FUNCTION_BLOCK FB_StackerLiftControl
VAR_INPUT
	FunctionData			: ST_FunctionData; 						// Function data
	ZoneData				: ST_ZoneData;
	EnableDrive				: BOOL;								//forks not moving	
	OrderPos				: E_StackerLiftPositions; 		// Order position of palletmagazine	
	LiftEncoderType			: BOOL;								// TRUE: Encoder is used for positioning, False: Inductive sensors is used
	SensorInputs			: ST_StackerLiftSensorInp;			// Lift sensor inputs
	ManualInputs			: ST_StackerLiftManualInp;			// Manual control inputs
	EncoderSettings			: ST_LSPM_LiftEncPos;			// Encoder configuration
	TimeoutValueLift		: TIME; 							// Timeout value for turning	
	
END_VAR

VAR_OUTPUT
	DriveUp					: BOOL; 							// Drive run command lift up
	DriveDown				: BOOL; 							// Drive run command lift down
	DriveCS					: BOOL; 							// Drive run command lift low speed
	EnableTransport			: BOOL;								// Enable transport
	ActualPosition			: E_StackerLiftPositions;		// The position of the lift
END_VAR

VAR_IN_OUT
	ErrorData 				: ST_ErrorDataSet; // Error data
END_VAR

VAR
	eState					: E_StackerLiftStates;
	eLastState				: E_StackerLiftStates;	
	TimerTimeoutLift		: TON;		
	TimerIdle				: TON := (PT:= T#500MS);  // delay setting EnableTransport until lift motor realy stopped
END_VAR


F_ResetError(
	Reset 	  := FALSE,
	ErrorData := ErrorData);


// Initialise variables	
DriveUp := FALSE;
DriveDown := FALSE;
EnableTransport := FALSE;	
TimerTimeoutLift.IN := FALSE;
TimerTimeoutLift.PT := TimeoutValueLift;
//ActualPosition := E_PositionsPalletMagazineForkLift.UNDEFINED;
ActualPosition 	:= _M_GetActualPosition(LiftEncoderType,SensorInputs,EncoderSettings,ErrorData);
 

CASE eState OF
	(*************************************************************************
	  Initialise
	*************************************************************************)	
	E_StackerLiftStates.INIT:
		DriveUp := FALSE;
		DriveDown := FALSE;
		DriveCS := FALSE;		
		EnableTransport := FALSE;	
	
		eLastState := eState;
		eState := E_StackerLiftStates.IDLE;
		
	(*************************************************************************
	  Error
	*************************************************************************)	
	E_StackerLiftStates.Error:

		IF NOT ManualInputs.SwitchManualAuto THEN
			eLastState := eState;
			eState := E_StackerLiftStates.MANUAL;

		// Acknowledge request error
		ELSIF ErrorData.ErrorType <> E_ErrorType.ERROR AND 
			FunctionData.ErrorData.Error.ErrorType <> E_ErrorType.ERROR AND ZoneData.ErrorData.ErrorState <> E_ErrorState.ERROR  THEN	
			eLastState := eState;
			eState := E_StackerLiftStates.Init;			
		END_IF	

	(*************************************************************************
	  Manual
	*************************************************************************)			
	E_StackerLiftStates.MANUAL:		
		IF ManualInputs.SwitchManualAuto THEN
			eLastState := eState;
			eState := E_StackerLiftStates.INIT;		
		ELSE
			_M_ManualMode(LiftEncoderType,SensorInputs,ManualInputs,EncoderSettings,ActualPosition);			
		END_IF
	(*************************************************************************
	  Idle
	*************************************************************************)		
	E_StackerLiftStates.IDLE:
		IF NOT ManualInputs.SwitchManualAuto THEN
			eLastState := eState;
			eState := E_StackerLiftStates.MANUAL;

		// If function is started and no error	
		ELSIF ((FunctionData.OperationState.eState = E_PositionState.STARTED OR FunctionData.OperationState.eState = E_PositionState.STOPPING) AND
		  	   FunctionData.ErrorData.Error.ErrorType <> E_ErrorType.ERROR AND ZoneData.ErrorData.ErrorState <> E_ErrorState.ERROR) THEN		  	
					
			DriveCS := FALSE;	
	
			IF OrderPos = E_StackerLiftPositions.DOWN THEN
				// When Lift is in position down (lowest position)
				IF ActualPosition = E_StackerLiftPositions.DOWN THEN
					EnableTransport := TimerIdle.Q;
				ELSIF(EnableDrive AND FunctionData.OperationState.eState = E_PositionState.STARTED) THEN //only start movment if group is started and not stopping
					eLastState := eState;
					eState := E_StackerLiftStates.LIFT_DOWN;
				END_IF
				
			ELSIF OrderPos = E_StackerLiftPositions.UP THEN
				// When lift is in upper position, second pallet lifted up
				IF ActualPosition = E_StackerLiftPositions.Up THEN
					EnableTransport := TimerIdle.Q;
				ELSIF(EnableDrive AND FunctionData.OperationState.eState = E_PositionState.STARTED) THEN //only start movment if group is started and not stopping
					eLastState := eState;
					eState := E_StackerLiftStates.LIFT_UP;
				END_IF
				
			ELSIF OrderPos = E_StackerLiftPositions.MIDDLE THEN
				// When lift is ordered to the middle position 
				IF ActualPosition = E_StackerLiftPositions.MIDDLE THEN
					EnableTransport := TimerIdle.Q;
				ELSIF(EnableDrive AND FunctionData.OperationState.eState = E_PositionState.STARTED) THEN //only start movment if group is started and not stopping
					IF( _M_DecideNextMovement(OrderPos,LiftEncoderType,SensorInputs,EncoderSettings) = E_StackerLiftStates.LIFT_MIDDLE_FROM_DOWN) THEN
						eLastState := eState;
						eState := E_StackerLiftStates.LIFT_MIDDLE_FROM_DOWN;
					ELSIF( _M_DecideNextMovement(OrderPos,LiftEncoderType,SensorInputs,EncoderSettings) = E_StackerLiftStates.LIFT_MIDDLE_FROM_UP) THEN
						eLastState := eState;
						eState := E_StackerLiftStates.LIFT_MIDDLE_FROM_UP;
					ELSE
						//can not decide next movment, since we dont know where we are
						F_SetError( ErrorType := E_ErrorType.ERROR, 
									ErrorParam := 'Middle position unknown.', //Can not decide next movment 
									ErrorMsg := E_ErrorConv.INCORRECT_SENSOR_SIGNAL, 
									ErrorData := ErrorData);
						
					END_IF
				END_IF			
			END_IF
		ELSE
			eLastState := eState;
			eState := E_StackerLiftStates.Error;		  
		END_IF	
	
	(*************************************************************************
	  Turn to ccw
	*************************************************************************)	
	E_StackerLiftStates.LIFT_DOWN:
		// If function is started or stopping and no error
		IF (FunctionData.OperationState.eState = E_PositionState.STARTED OR FunctionData.OperationState.eState = E_PositionState.STOPPING) AND
		  FunctionData.ErrorData.Error.ErrorType <> E_ErrorType.ERROR AND ZoneData.ErrorData.ErrorState <> E_ErrorState.ERROR THEN
			// Moving lift down until desired level is reached			
			TimerTimeoutLift.IN := TRUE;
			// If time is up
			IF TimerTimeoutLift.Q THEN
				DriveDown := FALSE;
				F_SetError(
					ErrorType := E_ErrorType.ERROR, 
					ErrorParam := 'Timeout Lifting Down', 
					ErrorMsg := E_ErrorConv.TIMEOUT_MOVEMENT, 
					ErrorData := ErrorData);
					
				eLastState := eState;
				eState := E_StackerLiftStates.Error;
			ELSIF(_M_DecideStopAndCreep(eState,LiftEncoderType,SensorInputs,EncoderSettings, ActualPosition,ErrorData,DriveCS)) THEN
				eLastState := eState;
				eState := E_StackerLiftStates.IDLE;			
			ELSIF EnableDrive THEN
				DriveDown := TRUE;
				//DriveCS := _M_DecideCreepSpeed(eState,LiftType,SensorInputs,EncoderSettings);		
			END_IF
		ELSE
			eLastState := eState;
			eState := E_StackerLiftStates.Error;			
		END_IF
		
	
	(*************************************************************************
	  Turn to cw
	*************************************************************************)		
	E_StackerLiftStates.LIFT_UP:
	
		IF (FunctionData.OperationState.eState = E_PositionState.STARTED OR FunctionData.OperationState.eState = E_PositionState.STOPPING) AND
		  FunctionData.ErrorData.Error.ErrorType <> E_ErrorType.ERROR AND ZoneData.ErrorData.ErrorState <> E_ErrorState.ERROR THEN
			// Moving lift up until desired level is reached
			TimerTimeoutLift.IN := TRUE;
				
			// If time is up
			IF TimerTimeoutLift.Q THEN
				DriveUp := FALSE;
				F_SetError(
					ErrorType := E_ErrorType.ERROR, 
					ErrorParam := 'Timeout Lifting Up', 
					ErrorMsg := E_ErrorConv.TIMEOUT_MOVEMENT, 
					ErrorData := ErrorData);
					
				eLastState := eState;
				eState := E_StackerLiftStates.Error;
			ELSIF(_M_DecideStopAndCreep(eState,LiftEncoderType,SensorInputs,EncoderSettings, ActualPosition,ErrorData,DriveCS)) THEN
				eLastState := eState;
				eState := E_StackerLiftStates.IDLE;
			ELSIF EnableDrive THEN
				DriveUp := TRUE;
				//DriveCS := _M_DecideCreepSpeed(eState,LiftType,SensorInputs,EncoderSettings);		
			END_IF		
		ELSE
			eLastState := eState;
			eState := E_StackerLiftStates.Error;			
		END_IF

	(*************************************************************************
	  Turn to middle from ccw
	*************************************************************************)
	E_StackerLiftStates.LIFT_MIDDLE_FROM_DOWN:
	
		IF (FunctionData.OperationState.eState = E_PositionState.STARTED OR FunctionData.OperationState.eState = E_PositionState.STOPPING) AND
		  FunctionData.ErrorData.Error.ErrorType <> E_ErrorType.ERROR AND ZoneData.ErrorData.ErrorState <> E_ErrorState.ERROR THEN			
			// Moving lift up to the middle poistition until desired level is reached
			TimerTimeoutLift.IN := TRUE;				
			// If time is up
			IF TimerTimeoutLift.Q THEN
				DriveUp := FALSE;
				F_SetError(
					ErrorType := E_ErrorType.ERROR, 
					ErrorParam := 'Timeout Lifting to Middle from Down', 
					ErrorMsg := E_ErrorConv.TIMEOUT_MOVEMENT, 
					ErrorData := ErrorData);
					
				eLastState := eState;
				eState := E_StackerLiftStates.Error;
			ELSIF(_M_DecideStopAndCreep(eState,LiftEncoderType,SensorInputs,EncoderSettings, ActualPosition,ErrorData,DriveCS)) THEN
				eLastState := eState;
				eState := E_StackerLiftStates.IDLE;
			ELSIF EnableDrive THEN
				DriveUp := TRUE;
				//DriveCS := _M_DecideCreepSpeed(eState,LiftType,SensorInputs,EncoderSettings);	
			END_IF

		ELSE
			eLastState := eState;
			eState := E_StackerLiftStates.Error;
		END_IF
		
	(*************************************************************************
	  Turn to middle from cw
	*************************************************************************)		
	E_StackerLiftStates.LIFT_MIDDLE_FROM_UP:
	
		IF (FunctionData.OperationState.eState = E_PositionState.STARTED OR FunctionData.OperationState.eState = E_PositionState.STOPPING) AND
		  FunctionData.ErrorData.Error.ErrorType <> E_ErrorType.ERROR AND ZoneData.ErrorData.ErrorState <> E_ErrorState.ERROR THEN			
			// Moving lift down to the middle poistition until desired level is reached
			TimerTimeoutLift.IN := TRUE;
			// If time is up
			IF TimerTimeoutLift.Q THEN
				DriveDown := FALSE;
				F_SetError(
					ErrorType := E_ErrorType.ERROR, 
					ErrorParam := 'Timeout Liftning to Middle from Up', 
					ErrorMsg := E_ErrorConv.TIMEOUT_MOVEMENT, 
					ErrorData := ErrorData);
					
				eLastState := eState;
				eState := E_StackerLiftStates.Error;
				
			ELSIF(_M_DecideStopAndCreep(eState,LiftEncoderType,SensorInputs,EncoderSettings, ActualPosition,ErrorData,DriveCS)) THEN
				eLastState := eState;
				eState := E_StackerLiftStates.IDLE;
			ELSIF EnableDrive THEN
				DriveDown := TRUE;
				//DriveCS := _M_DecideCreepSpeed(eState,LiftType,SensorInputs,EncoderSettings);	
			END_IF		
		ELSE
			eLastState := eState;
			eState := E_StackerLiftStates.Error;			
		END_IF
END_CASE

TimerTimeoutLift();
TimerIdle(IN := eState=E_StackerLiftStates.IDLE);

//When order pos is Middle, we need to determine if going to middle from above or from below
METHOD PRIVATE _M_DecideNextMovement : E_StackerLiftStates
VAR_INPUT
	OrderPos 				: E_StackerLiftPositions;
	LiftEncoderType			: BOOL;							// TRUE: Encoder is used for positioning, False: Inductive sensors is used
	SensorInputs			: ST_StackerLiftSensorInp;	
	EncoderSettings			: ST_LSPM_LiftEncPos;
END_VAR

IF( OrderPos <> E_StackerLiftPositions.MIDDLE) THEN
	_M_DecideNextMovement := E_StackerLiftStates.IDLE;
	RETURN;
END_IF


IF(NOT LiftEncoderType) THEN

	IF(SensorInputs.SensorPosDown OR (SensorInputs.SensorPosMiddleDown AND NOT SensorInputs.SensorPosMiddleUp)) THEN
		_M_DecideNextMovement := E_StackerLiftStates.LIFT_MIDDLE_FROM_DOWN;
	
	ELSIF(SensorInputs.SensorPosUp OR (SensorInputs.SensorPosMiddleUp AND NOT SensorInputs.SensorPosMiddleDown)) THEN
		_M_DecideNextMovement :=E_StackerLiftStates.LIFT_MIDDLE_FROM_UP;
	END_IF		
END_IF
		

IF(LiftEncoderType) THEN
	
	IF( SensorInputs.EncoderValue <= EncoderSettings.Middle) THEN		   
		_M_DecideNextMovement := E_StackerLiftStates.LIFT_MIDDLE_FROM_DOWN;
		
	ELSIF( SensorInputs.EncoderValue >= EncoderSettings.Middle) THEN		   
		_M_DecideNextMovement := E_StackerLiftStates.LIFT_MIDDLE_FROM_UP;	
	END_IF
	
END_IF
END_METHOD

//Check if the desired position is reached. 
//Check if creep speed conditions is met.
METHOD PRIVATE _M_DecideStopAndCreep : BOOL
VAR_INPUT
	State					: E_StackerLiftStates;
	LiftEncoderType			: BOOL;							// TRUE: Encoder is used for positioning, False: Inductive sensors is used
	SensorInputs			: ST_StackerLiftSensorInp;	
	EncoderSettings			: ST_LSPM_LiftEncPos;
	ActualPosition			: E_StackerLiftPositions;
END_VAR
VAR_IN_OUT	
	ErrorData 				: ST_ErrorDataSet; // Error data
	Creep					: BOOL;
END_VAR

//stop conditions are not the same as to determine the actual position

//Inductive sensor lift type
IF(NOT LiftEncoderType) THEN
	IF(State = E_StackerLiftStates.LIFT_DOWN) THEN
		_M_DecideStopAndCreep := SensorInputs.SensorPosDown;		
		Creep := SensorInputs.SensorPosDownCS OR SensorInputs.SensorPosDown;
		//Check that the lower lift position is equal to the definition of lift DOWN
		IF(_M_DecideStopAndCreep AND (ActualPosition <> E_StackerLiftPositions.DOWN)) THEN
			F_SetError(
						ErrorType := E_ErrorType.ERROR, 
						ErrorParam := 'Lift Lower position both sensors not detected', 
						ErrorMsg := E_ErrorConv.INCORRECT_SENSOR_SIGNAL, 
						ErrorData := ErrorData);
		END_IF
		
	END_IF
	
	IF(State = E_StackerLiftStates.LIFT_UP) THEN
		_M_DecideStopAndCreep := ActualPosition = E_StackerLiftPositions.UP;
		Creep := FALSE; //there is no creep speed sensor moving up		
	END_IF
	
	IF(State = E_StackerLiftStates.LIFT_MIDDLE_FROM_DOWN) THEN
		_M_DecideStopAndCreep := SensorInputs.SensorPosMiddleUp; //stop when middle up sensor is detected.
		Creep := SensorInputs.SensorPosMiddleDown;	 	
	
		IF(_M_DecideStopAndCreep AND (ActualPosition <> E_StackerLiftPositions.MIDDLE)) THEN
			F_SetError(
						ErrorType := E_ErrorType.ERROR, 
						ErrorParam := 'Lift middle position both sensors not detected', 
						ErrorMsg := E_ErrorConv.INCORRECT_SENSOR_SIGNAL, 
						ErrorData := ErrorData);
		END_IF
	END_IF
	
	IF(State = E_StackerLiftStates.LIFT_MIDDLE_FROM_UP) THEN
		_M_DecideStopAndCreep := SensorInputs.SensorPosMiddleDown;
		Creep := SensorInputs.SensorPosMiddleUp;
		IF(_M_DecideStopAndCreep AND (ActualPosition <> E_StackerLiftPositions.MIDDLE)) THEN
			F_SetError(
						ErrorType := E_ErrorType.ERROR, 
						ErrorParam := 'Both middle position sensors not detected', 
						ErrorMsg := E_ErrorConv.INCORRECT_SENSOR_SIGNAL, 
						ErrorData := ErrorData);
		END_IF	
	END_IF
	
END_IF


//Encoder lift type
IF(LiftEncoderType) THEN
	IF(State = E_StackerLiftStates.LIFT_DOWN) THEN
		_M_DecideStopAndCreep := (SensorInputs.EncoderValue <= EncoderSettings.Lower + EncoderSettings.Tolerance);
		Creep := Creep OR SensorInputs.EncoderValue <= EncoderSettings.Lower + EncoderSettings.CsWindow AND
				 		  SensorInputs.EncoderValue >= EncoderSettings.Lower - EncoderSettings.CsWindow;
		
		IF(_M_DecideStopAndCreep AND (ActualPosition <> E_StackerLiftPositions.DOWN)) THEN
			F_SetError(
						ErrorType := E_ErrorType.ERROR, 
						ErrorParam := 'Lift Lower positioning error', 
						ErrorMsg := E_ErrorConv.INCORRECT_SENSOR_SIGNAL, 
						ErrorData := ErrorData);
		END_IF
		
	END_IF
	
	IF(State = E_StackerLiftStates.LIFT_UP) THEN
		_M_DecideStopAndCreep := (SensorInputs.EncoderValue >= EncoderSettings.Upper - EncoderSettings.Tolerance);
		Creep := FALSE; //there is no creep speed window used moving up		
	END_IF
	
	IF(State = E_StackerLiftStates.LIFT_MIDDLE_FROM_DOWN) THEN
		_M_DecideStopAndCreep := (SensorInputs.EncoderValue >= EncoderSettings.Middle - EncoderSettings.Tolerance);
		Creep :=  Creep OR SensorInputs.EncoderValue >= EncoderSettings.Middle - EncoderSettings.CsWindow AND
				 		   SensorInputs.EncoderValue <= EncoderSettings.Middle + EncoderSettings.CsWindow;	
		IF(_M_DecideStopAndCreep AND (ActualPosition <> E_StackerLiftPositions.MIDDLE)) THEN
			F_SetError(
						ErrorType := E_ErrorType.ERROR, 
						ErrorParam := 'Lift middle position could not be determined', 
						ErrorMsg := E_ErrorConv.INCORRECT_SENSOR_SIGNAL, 
						ErrorData := ErrorData);
		END_IF
	END_IF
	
	IF(State = E_StackerLiftStates.LIFT_MIDDLE_FROM_UP) THEN
		_M_DecideStopAndCreep := (SensorInputs.EncoderValue <= EncoderSettings.Middle + EncoderSettings.Tolerance);
		Creep := Creep OR SensorInputs.EncoderValue <= EncoderSettings.Middle + EncoderSettings.CsWindow AND
				 		  SensorInputs.EncoderValue >= EncoderSettings.Middle - EncoderSettings.CsWindow;
		IF(_M_DecideStopAndCreep AND (ActualPosition <> E_StackerLiftPositions.MIDDLE)) THEN
			F_SetError(
						ErrorType := E_ErrorType.ERROR, 
						ErrorParam := 'Lift middle position could not be determined', 
						ErrorMsg := E_ErrorConv.INCORRECT_SENSOR_SIGNAL, 
						ErrorData := ErrorData);
		END_IF	
	END_IF

END_IF
END_METHOD

METHOD PRIVATE _M_GetActualPosition : E_StackerLiftPositions
VAR_INPUT	
	LiftEncoderType			: BOOL;							// TRUE: Encoder is used for positioning, False: Inductive sensors is used
	SensorInputs			: ST_StackerLiftSensorInp;	
	EncoderSettings			: ST_LSPM_LiftEncPos;
END_VAR
VAR_IN_OUT
	ErrorData 				: ST_ErrorDataSet; // Error data
END_VAR

_M_GetActualPosition := E_StackerLiftPositions.UNDEFINED;


//Inductive senor lift type
IF(NOT LiftEncoderType) THEN
	
	IF(SensorInputs.SensorPosDown AND SensorInputs.SensorPosDownCS) THEN
		_M_GetActualPosition := E_StackerLiftPositions.DOWN;
	ELSIF(SensorInputs.SensorPosUp) THEN
		_M_GetActualPosition := E_StackerLiftPositions.UP;		
	ELSIF(SensorInputs.SensorPosMiddleDown AND SensorInputs.SensorPosMiddleUp) THEN
		_M_GetActualPosition := E_StackerLiftPositions.MIDDLE;	
	END_IF
	
	
	// Sensor error check
	IF (SensorInputs.SensorPosDown AND SensorInputs.SensorPosUp) OR 
		(SensorInputs.SensorPosDown AND (SensorInputs.SensorPosMiddleDown AND SensorInputs.SensorPosMiddleUp)) OR 
		(SensorInputs.SensorPosUp AND (SensorInputs.SensorPosMiddleDown AND SensorInputs.SensorPosMiddleUp)) THEN			
			F_SetError(
				ErrorType := E_ErrorType.ERROR, 
				ErrorParam := 'Two position sensors active', 
				ErrorMsg := E_ErrorConv.INCORRECT_SENSOR_SIGNAL, 
				ErrorData := ErrorData);
	END_IF
	
END_IF




//Encoder lift type
IF(LiftEncoderType) THEN
	
	IF( (SensorInputs.EncoderValue <= EncoderSettings.Lower + EncoderSettings.Tolerance) AND
		(SensorInputs.EncoderValue >= EncoderSettings.Lower - EncoderSettings.Tolerance)) THEN
		_M_GetActualPosition := E_StackerLiftPositions.DOWN;
	
	ELSIF( (SensorInputs.EncoderValue <= EncoderSettings.Middle + EncoderSettings.Tolerance) AND
		   (SensorInputs.EncoderValue >= EncoderSettings.Middle - EncoderSettings.Tolerance)) THEN
		_M_GetActualPosition := E_StackerLiftPositions.MIDDLE;
		
	ELSIF( (SensorInputs.EncoderValue >= EncoderSettings.Upper - EncoderSettings.Tolerance) (*AND
		   (SensorInputs.EncoderValue <= EncoderSettings.Upper + EncoderSettings.PositioningTolerance)*)) THEN
		_M_GetActualPosition := E_StackerLiftPositions.UP;	
	END_IF
	
	
	IF( (SensorInputs.EncoderValue < EncoderSettings.LowerEndLimit) OR
		(SensorInputs.EncoderValue > EncoderSettings.UpperEndLimit)) THEN
	
		F_SetError(
				ErrorType := E_ErrorType.ERROR, 
				ErrorParam := 'Position outside valid range', 
				ErrorMsg := E_ErrorConv.INCORRECT_SENSOR_SIGNAL, 
				ErrorData := ErrorData);
	END_IF	
END_IF
END_METHOD

METHOD PRIVATE _M_ManualMode : BOOL
VAR_INPUT	
	LiftEncoderType			: BOOL;							// TRUE: Encoder is used for positioning, False: Inductive sensors is used
	SensorInputs			: ST_StackerLiftSensorInp;		// Lift sensor inputs
	ManualInputs			: ST_StackerLiftManualInp;		// Manual control inputs
	EncoderSettings			: ST_LSPM_LiftEncPos;		// Encoder configuration
	ActualPos				: E_StackerLiftPositions;	// Actual lift position
END_VAR
VAR_INST
	PositiveEdgeMan		: R_TRIG;
	ManualInPos				: BOOL;
END_VAR
VAR
		
	TempErrorData 			: ST_ErrorDataSet; // Temporary error data
	Creep					: BOOL;
	i						: E_StackerLiftStates;
END_VAR

// If down,middle or up positioin is reached, then the user must re-push the button in order to move lift up or down


PositiveEdgeMan(CLK := ActualPos=E_StackerLiftPositions.DOWN OR
					   ActualPos=E_StackerLiftPositions.MIDDLE OR
					   ActualPos=E_StackerLiftPositions.UP);
					   
   
IF PositiveEdgeMan.Q THEN 
	ManualInPos := TRUE;
ELSIF NOT ManualInputs.SwitchDriveUp AND NOT ManualInputs.SwitchDriveDown THEN 
	ManualInPos := FALSE;				
END_IF

DriveUp 	:= ManualInputs.SwitchDriveUp 	AND NOT ManualInPos;
DriveDown 	:= ManualInputs.SwitchDriveDown	AND NOT ManualInPos;
DriveCS		:= FALSE;

//set creep speed, check all possible modes

IF(ManualInputs.SwitchDriveDown) THEN
	_M_DecideStopAndCreep(
		State				:= E_StackerLiftStates.LIFT_DOWN, 
		LiftEncoderType		:= LiftEncoderType, 
		SensorInputs		:= SensorInputs, 
		EncoderSettings		:= EncoderSettings, 
		ActualPosition		:= ActualPos, 
		ErrorData			:= TempErrorData, 
		Creep				:= Creep);		
	DriveCS := DriveCS OR Creep;
	
	_M_DecideStopAndCreep(
		State				:= E_StackerLiftStates.LIFT_MIDDLE_FROM_UP, 
		LiftEncoderType		:= LiftEncoderType, 
		SensorInputs		:= SensorInputs, 
		EncoderSettings		:= EncoderSettings, 
		ActualPosition		:= ActualPos, 
		ErrorData			:= TempErrorData, 
		Creep				:= Creep);
		
	DriveCS := DriveCS OR Creep;
END_IF

IF(ManualInputs.SwitchDriveUp) THEN
	_M_DecideStopAndCreep(
		State				:= E_StackerLiftStates.LIFT_UP, 
		LiftEncoderType		:= LiftEncoderType, 
		SensorInputs		:= SensorInputs, 
		EncoderSettings		:= EncoderSettings, 
		ActualPosition		:= ActualPos, 
		ErrorData			:= TempErrorData, 
		Creep				:= Creep);		
	DriveCS := DriveCS OR Creep;
	
	_M_DecideStopAndCreep(
		State				:= E_StackerLiftStates.LIFT_MIDDLE_FROM_DOWN, 
		LiftEncoderType		:= LiftEncoderType, 
		SensorInputs		:= SensorInputs, 
		EncoderSettings		:= EncoderSettings, 
		ActualPosition		:= ActualPos, 
		ErrorData			:= TempErrorData, 
		Creep				:= Creep);
		
	DriveCS := DriveCS OR Creep;
END_IF
END_METHOD

END_FUNCTION_BLOCK

(* stored: Version 1.1.0.1, ProductVersion 3.1.4024.9
   POU FB_StackerLiftControl: Id {1d4af2ac-6fc6-4ae6-8e44-af88fed9850f}, SpecialFunc None
   Method _M_DecideNextMovement: Id {bb57207d-9cf4-486e-bc98-49471b29e42f}
   Method _M_DecideStopAndCreep: Id {77945a4b-e6b2-42dc-8f92-cc2d413640d9}
   Method _M_GetActualPosition: Id {4a678a2e-0ef6-48a6-9cf7-5b0734a1977b}
   Method _M_ManualMode: Id {d45e0872-89dd-40aa-ae10-99c188f53580} *)
